{attribute 'qualified_only'}
{attribute 'strict'}
TYPE E_ConnectSteps :
(
	//E_Connect_idle,
	//E_Connect_Start,
	//E_Connect_Wait,
	//E_Connect_DataExchange,
	//E_Connect_CloseStart,
	//E_Connect_CloseWait,
	//E_Connect_Error
	DUMMY
);
END_TYPE

(* stored: Version 1.1.0.1
   DUT E_ConnectSteps: Id {5f472d66-9de1-4737-9615-e7f06a4bd1ad} *)
